PROGRAM TEST_PROG
VAR
	BaseUnitTests : FB_BaseUnitTests;
	AxisBaseUnitTests : FB_Axis_BaseUnitTests;
	FakeAxisContractTests : FB_FakeAxis_BaseUnitTests;
	UtcClockTests : FB_UtcClockTests;
	PackMLBaseTests : FB_PackMLBaseTests;
	PackMLModeSetTests : FB_PackMLModeSetTests;
	ServiceBaseTests : FB_ServiceBaseTests;
	ServiceExecuteSubStateTests : FB_ServiceExecuteSubStateTests;
	CompositeServiceBaseTests : FB_CompositeServiceBaseTests;
	SetMaterialServiceTests : FB_SetMaterialServiceTests;
	ServiceCallerTests : FB_ServiceCallerTests;
	ServiceCoordinatorTests : FB_ServiceCoordinatorTests;
	ModuleAlarmManagerTests : FB_ModuleAlarmManagerTests;
	ModuleBaseTests : FB_ModuleBaseTests;
	ConfigValueSnapshotReaderTests : FB_ConfigValueSnapshotReaderTests;
	LinkVariableManagerTests : FB_LinkVariableManagerTests;
	ReferenceManagerTests : FB_ReferenceManagerTests;
	ModuleReferenceBindingContextTests : FB_ModuleReferenceBindingContextTests;
	ModuleTypeRegistryTests : FB_ModuleTypeRegistryTests;
	ModuleConfigurationManagerTests : FB_ModuleConfigurationManagerTests;
	ApplicationConfigRootTests : FB_ApplicationConfigRootTests;
END_VAR

// 上述 FB_TestSuite instances 會向 TcUnit 註冊；runner 每個週期統一驅動測試。
TcUnit.RUN();

END_PROGRAM

(* stored: Version 1.1.0.1, ProductVersion 3.1.4026.18
   POU TEST_PROG: Id {8ff9d161-157e-42ac-b3da-373105b7f816}, SpecialFunc None *)
